Fanuc TP program (LS listing): UP022.LS

/PROG  UP022
/ATTR
OWNER		= GME;
COMMENT		= "Soldadura Est.";
PROG_SIZE	= 16158;
CREATE		= DATE 17-04-05  TIME 12:29:44;
MODIFIED	= DATE 24-03-02  TIME 05:16:32;
FILE_NAME	= UP022;
VERSION		= 0;
LINE_COUNT	= 65;
MEMORY_SIZE	= 30858;
PROTECT		= READ_WRITE;
TCD:  STACK_SIZE	= 500,
      TASK_PRIORITY	= 50,
      TIME_SLICE	= 0,
      BUSY_LAMP_OFF	= 0,
      ABORT_REQUEST	= 0,
      PAUSE_REQUEST	= 0;
DEFAULT_GROUP	= 1,1,1,1,*;
CONTROL_CODE	= 00000001 00000000;
/APPL
/MN
   1:  UFRAME_NUM=1 ;
   2:  UTOOL_NUM=2 ;
   3:  PAYLOAD[2] ;
   4:J P[1] 100% CNT0 ACC100 TB    .10sec,P-SPS    ;
      1:  TC_ONLINE (ON) ;
      2:  DO[23]=(OFF) ;
      3:  DO[16]=(ON) ;
      4:  TIMER[4]=RESET ;
      5:  TIMER[4]=START ;
      6:  CALL MAKRO050    ;
      7:  !Lib. de Herramientas ;
      8:  DO[80]=ON ;
      9:  DO[79]=ON ;
     10:  DO[78]=OFF ;
     11:  DO[77]=OFF ;
     12:  DO[76]=ON ;
     13:  DO[74]=OFF ;
     14:  !Lib. de Anticolisiones ;
     15:  DO[43]=ON ;
     16:  DO[44]=ON ;
     17:  DO[45]=ON ;
     18:  DO[46]=ON ;
     19:  DO[47]=ON ;
     20:  DO[48]=ON ;
     21:  !Apagar Pos. Base ;
     22:  DO[15]=OFF ;
     23:  !Robot en Trayectoria ;
     24:  DO[16]=ON ;
     25:  !Basculante 1 en Pos. de Reposo ;
     26:  IF (!DI[842] AND DO[12]),CALL MAKRO072 ;
     27:  WAIT (M[96])    ;
     28:  WAIT (DI[23])    ;
     29:  DO[23]=ON ;
     30:  TC_ONLINE (M[1] AND M[30] AND M[31] AND M[34] AND M[95] AND M[96]) ;
       ------ ;
   5:J P[2] 100% CNT100 ACC100 TB   0.00sec,P-SPS    ;
      1:  TC_ONLINE (M[1] AND M[30] AND M[31] AND M[34] AND M[95] AND M[96]) ;
       ------ ;
   6:J P[3] 100% CNT100 ACC100 TB   0.00sec,P-SPS    ;
      1:  TC_ONLINE (M[1] AND M[30] AND M[31] AND M[34] AND M[95] AND M[96]) ;
       ------ ;
   7:J P[4] 100% CNT100 ACC100 TB   0.00sec,P-SPS    ;
      1:  TC_ONLINE (M[1] AND M[30] AND M[31] AND M[34] AND M[95] AND M[96]) ;
       ------ ;
   8:  !5qa802035b_007_gps0005_L ;
   9:  !Punto de Sol. No. 10044 ;
  10:J P[5] 100% CNT0 ACC100 TB    .10sec,P-SPS Offset,PR[11]    ;
      1:  TC_ONLINE (ON) ;
      2:  DO[23]=(OFF) ;
      3:  WAIT (!DI[16] AND DI[23])    ;
      4:  CALL VW_USER(Basic1,EZSP,Nr1,ProgNr=99, , ,S-Punkt=10044,Fzg_Typ=7,EIN/AUS=ON) ;
      5:  GO[2]=(R[197]+10) ;
      6:  WAIT (!DI[129] OR DI[26])    ;
      7:  CALL MAKRO080    ;
      8:  WAIT (DI[23])    ;
      9:  DO[23]=(ON) ;
     10:  TC_ONLINE (M[1] AND M[30] AND M[31] AND M[34] AND M[95] AND M[96]) ;
       ------ ;
  11:J P[6] 100% CNT100 ACC100 TB   0.00sec,P-SPS    ;
      1:  TC_ONLINE (M[1] AND M[30] AND M[31] AND M[34] AND M[95] AND M[96]) ;
       ------ ;
  12:J P[7] 100% CNT100 ACC100 TB   0.00sec,P-SPS    ;
      1:  TC_ONLINE (M[1] AND M[30] AND M[31] AND M[34] AND M[95] AND M[96]) ;
       ------ ;
  13:J P[8] 100% CNT100 ACC100 TB   0.00sec,P-SPS    ;
      1:  TC_ONLINE (M[1] AND M[30] AND M[31] AND M[34] AND M[95] AND M[96]) ;
       ------ ;
  14:J P[9] 100% CNT100 ACC100 TB   0.00sec,P-SPS    ;
      1:  TC_ONLINE (M[1] AND M[30] AND M[31] AND M[34] AND M[95] AND M[96]) ;
       ------ ;
  15:  !5qa802035b_007_gps0007_L ;
  16:  !Punto de Sol. No. 10045 ;
  17:J P[10] 100% CNT0 ACC100 TB    .10sec,P-SPS Offset,PR[11]    ;
      1:  TC_ONLINE (ON) ;
      2:  DO[23]=(OFF) ;
      3:  WAIT (!DI[16] AND DI[23])    ;
      4:  CALL VW_USER(Basic1,EZSP,Nr1,ProgNr=99, , ,S-Punkt=10045,Fzg_Typ=7,EIN/AUS=ON) ;
      5:  GO[2]=(R[197]) ;
      6:  WAIT (!DI[129] OR DI[26])    ;
      7:  CALL MAKRO080    ;
      8:  WAIT (DI[23])    ;
      9:  DO[23]=(ON) ;
     10:  TC_ONLINE (M[1] AND M[30] AND M[31] AND M[34] AND M[95] AND M[96]) ;
       ------ ;
  18:J P[11] 100% CNT100 ACC100 TB   0.00sec,P-SPS    ;
      1:  TC_ONLINE (M[1] AND M[30] AND M[31] AND M[34] AND M[95] AND M[96]) ;
       ------ ;
  19:  !5qa802035b_023_xps0004_L ;
  20:  !Punto de Sol. No. 10046 ;
  21:J P[12] 100% CNT0 ACC100 TB    .10sec,P-SPS Offset,PR[11]    ;
      1:  TC_ONLINE (ON) ;
      2:  DO[23]=(OFF) ;
      3:  WAIT (!DI[16] AND DI[23])    ;
      4:  CALL VW_USER(Basic1,EZSP,Nr1,ProgNr=99, , ,S-Punkt=10046,Fzg_Typ=7,EIN/AUS=ON) ;
      5:  GO[2]=(R[197]+5) ;
      6:  WAIT (!DI[129] OR DI[26])    ;
      7:  CALL MAKRO080    ;
      8:  WAIT (DI[23])    ;
      9:  DO[23]=(ON) ;
     10:  TC_ONLINE (M[1] AND M[30] AND M[31] AND M[34] AND M[95] AND M[96]) ;
       ------ ;
  22:J P[13] 100% CNT100 ACC100 TB   0.00sec,P-SPS    ;
      1:  TC_ONLINE (M[1] AND M[30] AND M[31] AND M[34] AND M[95] AND M[96]) ;
       ------ ;
  23:J P[14] 100% CNT100 ACC100 TB   0.00sec,P-SPS    ;
      1:  TC_ONLINE (M[1] AND M[30] AND M[31] AND M[34] AND M[95] AND M[96]) ;
       ------ ;
  24:J P[15] 100% CNT100 ACC100 TB   0.00sec,P-SPS    ;
      1:  TC_ONLINE (M[1] AND M[30] AND M[31] AND M[34] AND M[95] AND M[96]) ;
       ------ ;
  25:J P[16] 100% CNT100 ACC100 TB   0.00sec,P-SPS    ;
      1:  TC_ONLINE (M[1] AND M[30] AND M[31] AND M[34] AND M[95] AND M[96]) ;
       ------ ;
  26:J P[17] 100% CNT100 ACC100 TB   0.00sec,P-SPS    ;
      1:  TC_ONLINE (M[1] AND M[30] AND M[31] AND M[34] AND M[95] AND M[96]) ;
       ------ ;
  27:J P[18] 100% CNT100 ACC100 TB   0.00sec,P-SPS    ;
      1:  TC_ONLINE (M[1] AND M[30] AND M[31] AND M[34] AND M[95] AND M[96]) ;
       ------ ;
  28:J P[19] 100% CNT100 ACC100 TB   0.00sec,P-SPS    ;
      1:  TC_ONLINE (M[1] AND M[30] AND M[31] AND M[34] AND M[95] AND M[96]) ;
       ------ ;
  29:  !5qa802035b_013_nps0004_L ;
  30:  !Punto de Sol. No. 10053 ;
  31:J P[20] 100% CNT0 ACC100 TB    .10sec,P-SPS Offset,PR[11]    ;
      1:  TC_ONLINE (ON) ;
      2:  DO[23]=(OFF) ;
      3:  WAIT (!DI[16] AND DI[23])    ;
      4:  CALL VW_USER(Basic1,EZSP,Nr1,ProgNr=99, , ,S-Punkt=10053,Fzg_Typ=7,EIN/AUS=ON) ;
      5:  GO[2]=(R[197]) ;
      6:  WAIT (!DI[129] OR DI[26])    ;
      7:  CALL MAKRO080    ;
      8:  WAIT (DI[23])    ;
      9:  DO[23]=(ON) ;
     10:  TC_ONLINE (M[1] AND M[30] AND M[31] AND M[34] AND M[95] AND M[96]) ;
       ------ ;
  32:  !5qa802035b_013_nps0003_L ;
  33:  !Punto de Sol. No. 10052 ;
  34:J P[21] 100% CNT0 ACC100 TB    .10sec,P-SPS Offset,PR[11]    ;
      1:  TC_ONLINE (ON) ;
      2:  DO[23]=(OFF) ;
      3:  WAIT (!DI[16] AND DI[23])    ;
      4:  CALL VW_USER(Basic1,EZSP,Nr1,ProgNr=99, , ,S-Punkt=10052,Fzg_Typ=7,EIN/AUS=ON) ;
      5:  GO[2]=(R[197]+10) ;
      6:  WAIT (!DI[129] OR DI[26])    ;
      7:  CALL MAKRO080    ;
      8:  WAIT (DI[23])    ;
      9:  DO[23]=(ON) ;
     10:  TC_ONLINE (M[1] AND M[30] AND M[31] AND M[34] AND M[95] AND M[96]) ;
       ------ ;
  35:J P[22] 100% CNT100 ACC100 TB   0.00sec,P-SPS    ;
      1:  TC_ONLINE (M[1] AND M[30] AND M[31] AND M[34] AND M[95] AND M[96]) ;
       ------ ;
  36:J P[23] 100% CNT100 ACC100 TB   0.00sec,P-SPS    ;
      1:  TC_ONLINE (M[1] AND M[30] AND M[31] AND M[34] AND M[95] AND M[96]) ;
       ------ ;
  37:  !5qa802035b_029_adps0008_L ;
  38:  !Punto de Sol. No. 10051 ;
  39:J P[24] 100% CNT0 ACC100 TB    .10sec,P-SPS Offset,PR[11]    ;
      1:  TC_ONLINE (ON) ;
      2:  DO[23]=(OFF) ;
      3:  WAIT (!DI[16] AND DI[23])    ;
      4:  CALL VW_USER(Basic1,EZSP,Nr1,ProgNr=99, , ,S-Punkt=10051,Fzg_Typ=7,EIN/AUS=ON) ;
      5:  GO[2]=(R[197]) ;
      6:  WAIT (!DI[129] OR DI[26])    ;
      7:  CALL MAKRO080    ;
      8:  WAIT (DI[23])    ;
      9:  DO[23]=(ON) ;
     10:  TC_ONLINE (M[1] AND M[30] AND M[31] AND M[34] AND M[95] AND M[96]) ;
       ------ ;
  40:J P[25] 100% CNT100 ACC100 TB   0.00sec,P-SPS    ;
      1:  TC_ONLINE (M[1] AND M[30] AND M[31] AND M[34] AND M[95] AND M[96]) ;
       ------ ;
  41:  !5qa802035b_029_adps0009_L ;
  42:  !Punto de Sol. No. 10050 ;
  43:J P[26] 100% CNT0 ACC100 TB    .10sec,P-SPS Offset,PR[11]    ;
      1:  TC_ONLINE (ON) ;
      2:  DO[23]=(OFF) ;
      3:  WAIT (!DI[16] AND DI[23])    ;
      4:  CALL VW_USER(Basic1,EZSP,Nr1,ProgNr=99, , ,S-Punkt=10050,Fzg_Typ=7,EIN/AUS=ON) ;
      5:  GO[2]=(R[197]) ;
      6:  WAIT (!DI[129] OR DI[26])    ;
      7:  CALL MAKRO080    ;
      8:  WAIT (DI[23])    ;
      9:  DO[23]=(ON) ;
     10:  TC_ONLINE (M[1] AND M[30] AND M[31] AND M[34] AND M[95] AND M[96]) ;
       ------ ;
  44:  !5qa802035b_029_adps0005_L ;
  45:  !Punto de Sol. No. 10049 ;
  46:J P[27] 100% CNT0 ACC100 TB    .10sec,P-SPS Offset,PR[11]    ;
      1:  TC_ONLINE (ON) ;
      2:  DO[23]=(OFF) ;
      3:  WAIT (!DI[16] AND DI[23])    ;
      4:  CALL VW_USER(Basic1,EZSP,Nr1,ProgNr=99, , ,S-Punkt=10049,Fzg_Typ=7,EIN/AUS=ON) ;
      5:  GO[2]=(R[197]) ;
      6:  WAIT (!DI[129] OR DI[26])    ;
      7:  CALL MAKRO080    ;
      8:  WAIT (DI[23])    ;
      9:  DO[23]=(ON) ;
     10:  TC_ONLINE (M[1] AND M[30] AND M[31] AND M[34] AND M[95] AND M[96]) ;
       ------ ;
  47:J P[28] 100% CNT100 ACC100 TB   0.00sec,P-SPS    ;
      1:  TC_ONLINE (M[1] AND M[30] AND M[31] AND M[34] AND M[95] AND M[96]) ;
       ------ ;
  48:  !5qa802035b_013_nps0002_L ;
  49:  !Punto de Sol. No. 10048 ;
  50:J P[29] 100% CNT0 ACC100 TB    .10sec,P-SPS Offset,PR[11]    ;
      1:  TC_ONLINE (ON) ;
      2:  DO[23]=(OFF) ;
      3:  WAIT (!DI[16] AND DI[23])    ;
      4:  CALL VW_USER(Basic1,EZSP,Nr1,ProgNr=99, , ,S-Punkt=10048,Fzg_Typ=7,EIN/AUS=ON) ;
      5:  GO[2]=(R[197]) ;
      6:  WAIT (!DI[129] OR DI[26])    ;
      7:  CALL MAKRO080    ;
      8:  WAIT (DI[23])    ;
      9:  DO[23]=(ON) ;
     10:  TC_ONLINE (M[1] AND M[30] AND M[31] AND M[34] AND M[95] AND M[96]) ;
       ------ ;
  51:  !5qa802035b_013_nps0001_L ;
  52:  !Punto de Sol. No. 10047 ;
  53:J P[30] 100% CNT0 ACC100 TB    .10sec,P-SPS Offset,PR[11]    ;
      1:  TC_ONLINE (ON) ;
      2:  DO[23]=(OFF) ;
      3:  WAIT (!DI[16] AND DI[23])    ;
      4:  CALL VW_USER(Basic1,EZSP,Nr1,ProgNr=99, , ,S-Punkt=10047,Fzg_Typ=7,EIN/AUS=ON) ;
      5:  GO[2]=(R[197]) ;
      6:  WAIT (!DI[129] OR DI[26])    ;
      7:  CALL MAKRO080    ;
      8:  WAIT (DI[23])    ;
      9:  DO[23]=(ON) ;
     10:  TC_ONLINE (M[1] AND M[30] AND M[31] AND M[34] AND M[95] AND M[96]) ;
       ------ ;
  54:J P[31] 100% CNT100 ACC100 TB   0.00sec,P-SPS    ;
      1:  TC_ONLINE (M[1] AND M[30] AND M[31] AND M[34] AND M[95] AND M[96]) ;
       ------ ;
  55:J P[32] 100% CNT100 ACC100 TB   0.00sec,P-SPS    ;
      1:  TC_ONLINE (M[1] AND M[30] AND M[31] AND M[34] AND M[95] AND M[96]) ;
       ------ ;
  56:J P[33] 100% CNT100 ACC100 TB   0.00sec,P-SPS    ;
      1:  TC_ONLINE (M[1] AND M[30] AND M[31] AND M[34] AND M[95] AND M[96]) ;
       ------ ;
  57:J P[34] 100% CNT100 ACC100 TB   0.00sec,P-SPS    ;
      1:  TC_ONLINE (M[1] AND M[30] AND M[31] AND M[34] AND M[95] AND M[96]) ;
       ------ ;
  58:J P[35] 100% CNT100 ACC100 TB   0.00sec,P-SPS    ;
      1:  TC_ONLINE (M[1] AND M[30] AND M[31] AND M[34] AND M[95] AND M[96]) ;
       ------ ;
  59:  !5qa802035b_007_gps0003_L ;
  60:  !Punto de Sol. No. 10054 ;
  61:  !Fin de Trabajo 2 ;
  62:J P[36] 100% CNT0 ACC100 TB    .10sec,P-SPS Offset,PR[11]    ;
      1:  TC_ONLINE (ON) ;
      2:  DO[23]=(OFF) ;
      3:  WAIT (!DI[16] AND DI[23])    ;
      4:  CALL VW_USER(Basic1,EZSP,Nr1,ProgNr=99, , ,S-Punkt=10054,Fzg_Typ=7,EIN/AUS=ON) ;
      5:  GO[2]=(R[197]) ;
      6:  WAIT (!DI[129] OR DI[26])    ;
      7:  CALL MAKRO080    ;
      8:  IF (!DI[145] AND !DI[129]),CALL MAKRO002 ;
      9:  WAIT (DI[23])    ;
     10:  DO[23]=(ON) ;
     11:  TC_ONLINE (M[1] AND M[30] AND M[31] AND M[34] AND M[95] AND M[96]) ;
       ------ ;
  63:J P[37] 100% CNT100 ACC100 TB   0.00sec,P-SPS    ;
      1:  TC_ONLINE (M[1] AND M[30] AND M[31] AND M[34] AND M[95] AND M[96]) ;
       ------ ;
  64:J P[38] 100% CNT100 ACC100 TB   0.00sec,P-SPS    ;
      1:  TC_ONLINE (M[1] AND M[30] AND M[31] AND M[34] AND M[95] AND M[96]) ;
       ------ ;
  65:J P[39] 100% CNT0 ACC100 TB    .10sec,P-SPS    ;
      1:  TC_ONLINE (ON) ;
      2:  DO[23]=(OFF) ;
      3:  TIMER[4]=STOP ;
      4:  WAIT (DI[23])    ;
      5:  CALL VW_USER(Basic1,EZSP,Nr1 Service,ProgNr=31, , ,S-Punkt=31, ,EIN/AUS=1) ;
      6:  DO[23]=(ON) ;
      7:  TC_ONLINE (M[1] AND M[30] AND M[31] AND M[34] AND M[95] AND M[96]) ;
       ------ ;
/POS
P[1]{
   GP1:
	UF : 1, UT : 2,		CONFIG : 'N U T, 0, 0, 0',
	RX =  1133.105  mm,	RY =   304.802  mm,	RZ =  -956.232  mm,
	RW =    13.347 deg,	RP =    14.205 deg,	RR =   -95.327 deg
   GP2:
	UF : 1, UT : 2,
	J1=   100.000  mm
   GP3:
	UF : 1, UT : 2,
	J1=     0.000  mm
   GP4:
	UF : 1, UT : 2,
	J1=     0.000  mm
};
P[2]{
   GP1:
	UF : 1, UT : 2,		CONFIG : 'N U T, 0, 0, 0',
	RX =    66.244  mm,	RY = -1097.752  mm,	RZ =  -631.601  mm,
	RW =     4.264 deg,	RP =    -9.468 deg,	RR =  -138.417 deg
   GP2:
	UF : 1, UT : 2,
	J1=   120.000  mm
   GP3:
	UF : 1, UT : 2,
	J1=     0.000  mm
   GP4:
	UF : 1, UT : 2,
	J1=     0.000  mm
};
P[3]{
   GP1:
	UF : 1, UT : 2,		CONFIG : 'F U T, 0, 0, 0',
	RX =  -363.159  mm,	RY =  -637.383  mm,	RZ =   295.420  mm,
	RW =   171.646 deg,	RP =   -81.600 deg,	RR =    73.386 deg
   GP2:
	UF : 1, UT : 2,
	J1=   100.000  mm
   GP3:
	UF : 1, UT : 2,
	J1=     0.000  mm
   GP4:
	UF : 1, UT : 2,
	J1=     0.000  mm
};
P[4]{
   GP1:
	UF : 1, UT : 2,		CONFIG : 'F U T, 0, 0, 0',
	RX =  -355.700  mm,	RY =  -477.893  mm,	RZ =   268.172  mm,
	RW =   171.646 deg,	RP =   -81.600 deg,	RR =    73.385 deg
   GP2:
	UF : 1, UT : 2,
	J1=   100.000  mm
   GP3:
	UF : 1, UT : 2,
	J1=     0.000  mm
   GP4:
	UF : 1, UT : 2,
	J1=     0.000  mm
};
P[5]{
   GP1:
	UF : 1, UT : 2,		CONFIG : 'F U T, 0, 0, 0',
	RX =  -357.224  mm,	RY =  -466.560  mm,	RZ =   272.864  mm,
	RW =   169.052 deg,	RP =   -83.613 deg,	RR =    76.002 deg
   GP2:
	UF : 1, UT : 2,
	J1=    30.200  mm
   GP3:
	UF : 1, UT : 2,
	J1=     0.000  mm
   GP4:
	UF : 1, UT : 2,
	J1=     0.000  mm
};
P[6]{
   GP1:
	UF : 1, UT : 2,		CONFIG : 'F U T, 0, 0, 0',
	RX =  -359.183  mm,	RY =  -476.278  mm,	RZ =   268.090  mm,
	RW =   171.646 deg,	RP =   -81.600 deg,	RR =    73.386 deg
   GP2:
	UF : 1, UT : 2,
	J1=   100.000  mm
   GP3:
	UF : 1, UT : 2,
	J1=     0.000  mm
   GP4:
	UF : 1, UT : 2,
	J1=     0.000  mm
};
P[7]{
   GP1:
	UF : 1, UT : 2,		CONFIG : 'F U T, 0, 0, 0',
	RX =  -362.737  mm,	RY =  -548.013  mm,	RZ =   274.263  mm,
	RW =   171.645 deg,	RP =   -81.600 deg,	RR =    73.386 deg
   GP2:
	UF : 1, UT : 2,
	J1=   100.000  mm
   GP3:
	UF : 1, UT : 2,
	J1=     0.000  mm
   GP4:
	UF : 1, UT : 2,
	J1=     0.000  mm
};
P[8]{
   GP1:
	UF : 1, UT : 2,		CONFIG : 'F U T, 0, 0, 0',
	RX =  -129.372  mm,	RY =  -655.590  mm,	RZ =   283.757  mm,
	RW =   171.646 deg,	RP =   -81.600 deg,	RR =    73.386 deg
   GP2:
	UF : 1, UT : 2,
	J1=   100.000  mm
   GP3:
	UF : 1, UT : 2,
	J1=     0.000  mm
   GP4:
	UF : 1, UT : 2,
	J1=     0.000  mm
};
P[9]{
   GP1:
	UF : 1, UT : 2,		CONFIG : 'F U T, 0, 0, 0',
	RX =  -130.559  mm,	RY =  -455.743  mm,	RZ =   264.260  mm,
	RW =   177.915 deg,	RP =   -81.600 deg,	RR =    73.387 deg
   GP2:
	UF : 1, UT : 2,
	J1=   100.000  mm
   GP3:
	UF : 1, UT : 2,
	J1=     0.000  mm
   GP4:
	UF : 1, UT : 2,
	J1=     0.000  mm
};
P[10]{
   GP1:
	UF : 1, UT : 2,		CONFIG : 'F U T, 0, 0, 0',
	RX =  -129.044  mm,	RY =  -454.645  mm,	RZ =   269.211  mm,
	RW =   177.993 deg,	RP =   -81.609 deg,	RR =    73.315 deg
   GP2:
	UF : 1, UT : 2,
	J1=    27.704  mm
   GP3:
	UF : 1, UT : 2,
	J1=     0.000  mm
   GP4:
	UF : 1, UT : 2,
	J1=     0.000  mm
};
P[11]{
   GP1:
	UF : 1, UT : 2,		CONFIG : 'F U T, 0, 0, 0',
	RX =   -90.615  mm,	RY =  -443.457  mm,	RZ =   251.615  mm,
	RW =  -142.266 deg,	RP =   -79.369 deg,	RR =    33.067 deg
   GP2:
	UF : 1, UT : 2,
	J1=    40.000  mm
   GP3:
	UF : 1, UT : 2,
	J1=     0.000  mm
   GP4:
	UF : 1, UT : 2,
	J1=     0.000  mm
};
P[12]{
   GP1:
	UF : 1, UT : 2,		CONFIG : 'F U T, 0, 0, 0',
	RX =   -68.121  mm,	RY =  -445.925  mm,	RZ =   268.522  mm,
	RW =  -161.036 deg,	RP =   -72.891 deg,	RR =    52.407 deg
   GP2:
	UF : 1, UT : 2,
	J1=    22.000  mm
   GP3:
	UF : 1, UT : 2,
	J1=     0.000  mm
   GP4:
	UF : 1, UT : 2,
	J1=     0.000  mm
};
P[13]{
   GP1:
	UF : 1, UT : 2,		CONFIG : 'F U T, 0, 0, 0',
	RX =   -75.083  mm,	RY =  -452.168  mm,	RZ =   267.964  mm,
	RW =  -166.090 deg,	RP =   -74.801 deg,	RR =    57.641 deg
   GP2:
	UF : 1, UT : 2,
	J1=   100.000  mm
   GP3:
	UF : 1, UT : 2,
	J1=     0.000  mm
   GP4:
	UF : 1, UT : 2,
	J1=     0.000  mm
};
P[14]{
   GP1:
	UF : 1, UT : 2,		CONFIG : 'F U T, 0, 0, 0',
	RX =  -106.428  mm,	RY =  -546.571  mm,	RZ =   283.041  mm,
	RW =  -166.090 deg,	RP =   -74.801 deg,	RR =    57.641 deg
   GP2:
	UF : 1, UT : 2,
	J1=   100.000  mm
   GP3:
	UF : 1, UT : 2,
	J1=     0.000  mm
   GP4:
	UF : 1, UT : 2,
	J1=     0.000  mm
};
P[15]{
   GP1:
	UF : 1, UT : 2,		CONFIG : 'F U T, 0, 0, 0',
	RX =   -58.763  mm,	RY =  -675.997  mm,	RZ =   305.810  mm,
	RW =  -154.703 deg,	RP =   -81.518 deg,	RR =    46.029 deg
   GP2:
	UF : 1, UT : 2,
	J1=   100.000  mm
   GP3:
	UF : 1, UT : 2,
	J1=     0.000  mm
   GP4:
	UF : 1, UT : 2,
	J1=     0.000  mm
};
P[16]{
   GP1:
	UF : 1, UT : 2,		CONFIG : 'F U T, 0, 0, 0',
	RX =   167.422  mm,	RY =  -755.632  mm,	RZ =   268.835  mm,
	RW =  -117.579 deg,	RP =   -78.602 deg,	RR =     8.529 deg
   GP2:
	UF : 1, UT : 2,
	J1=   100.000  mm
   GP3:
	UF : 1, UT : 2,
	J1=     0.000  mm
   GP4:
	UF : 1, UT : 2,
	J1=     0.000  mm
};
P[17]{
   GP1:
	UF : 1, UT : 2,		CONFIG : 'F U T, 0, 0, 0',
	RX =   224.739  mm,	RY =  -491.620  mm,	RZ =   -22.031  mm,
	RW =  -102.440 deg,	RP =   -64.865 deg,	RR =    -7.291 deg
   GP2:
	UF : 1, UT : 2,
	J1=   100.000  mm
   GP3:
	UF : 1, UT : 2,
	J1=     0.000  mm
   GP4:
	UF : 1, UT : 2,
	J1=     0.000  mm
};
P[18]{
   GP1:
	UF : 1, UT : 2,		CONFIG : 'F U T, 0, 0, 0',
	RX =   186.154  mm,	RY =  -445.858  mm,	RZ =     4.056  mm,
	RW =  -100.027 deg,	RP =   -58.299 deg,	RR =   -10.029 deg
   GP2:
	UF : 1, UT : 2,
	J1=   100.000  mm
   GP3:
	UF : 1, UT : 2,
	J1=     0.000  mm
   GP4:
	UF : 1, UT : 2,
	J1=     0.000  mm
};
P[19]{
   GP1:
	UF : 1, UT : 2,		CONFIG : 'F U T, 0, 0, 0',
	RX =   173.095  mm,	RY =  -434.006  mm,	RZ =    19.013  mm,
	RW =  -106.388 deg,	RP =   -56.239 deg,	RR =    -2.521 deg
   GP2:
	UF : 1, UT : 2,
	J1=   100.000  mm
   GP3:
	UF : 1, UT : 2,
	J1=     0.000  mm
   GP4:
	UF : 1, UT : 2,
	J1=     0.000  mm
};
P[20]{
   GP1:
	UF : 1, UT : 2,		CONFIG : 'F U T, 0, 0, 0',
	RX =   175.846  mm,	RY =  -432.191  mm,	RZ =    12.536  mm,
	RW =  -108.251 deg,	RP =   -55.844 deg,	RR =     -.274 deg
   GP2:
	UF : 1, UT : 2,
	J1=    22.000  mm
   GP3:
	UF : 1, UT : 2,
	J1=     0.000  mm
   GP4:
	UF : 1, UT : 2,
	J1=     0.000  mm
};
P[21]{
   GP1:
	UF : 1, UT : 2,		CONFIG : 'F U T, 0, 0, 0',
	RX =   165.490  mm,	RY =  -431.087  mm,	RZ =    21.456  mm,
	RW =  -105.966 deg,	RP =   -56.296 deg,	RR =    -2.622 deg
   GP2:
	UF : 1, UT : 2,
	J1=    20.700  mm
   GP3:
	UF : 1, UT : 2,
	J1=     0.000  mm
   GP4:
	UF : 1, UT : 2,
	J1=     0.000  mm
};
P[22]{
   GP1:
	UF : 1, UT : 2,		CONFIG : 'F U T, 0, 0, 0',
	RX =   154.830  mm,	RY =  -426.794  mm,	RZ =    23.878  mm,
	RW =  -103.158 deg,	RP =   -56.239 deg,	RR =    -2.521 deg
   GP2:
	UF : 1, UT : 2,
	J1=    30.000  mm
   GP3:
	UF : 1, UT : 2,
	J1=     0.000  mm
   GP4:
	UF : 1, UT : 2,
	J1=     0.000  mm
};
P[23]{
   GP1:
	UF : 1, UT : 2,		CONFIG : 'F U T, 0, 0, 0',
	RX =   126.370  mm,	RY =  -417.423  mm,	RZ =    43.158  mm,
	RW =   -98.232 deg,	RP =   -56.239 deg,	RR =    -2.521 deg
   GP2:
	UF : 1, UT : 2,
	J1=    19.500  mm
   GP3:
	UF : 1, UT : 2,
	J1=     0.000  mm
   GP4:
	UF : 1, UT : 2,
	J1=     0.000  mm
};
P[24]{
   GP1:
	UF : 1, UT : 2,		CONFIG : 'F U T, 0, 0, 0',
	RX =   124.011  mm,	RY =  -422.950  mm,	RZ =    44.190  mm,
	RW =  -102.498 deg,	RP =   -54.643 deg,	RR =     2.578 deg
   GP2:
	UF : 1, UT : 2,
	J1=    22.000  mm
   GP3:
	UF : 1, UT : 2,
	J1=     0.000  mm
   GP4:
	UF : 1, UT : 2,
	J1=     0.000  mm
};
P[25]{
   GP1:
	UF : 1, UT : 2,		CONFIG : 'F U T, 0, 0, 0',
	RX =   107.911  mm,	RY =  -418.925  mm,	RZ =    49.571  mm,
	RW =   -97.335 deg,	RP =   -56.035 deg,	RR =     -.254 deg
   GP2:
	UF : 1, UT : 2,
	J1=    21.400  mm
   GP3:
	UF : 1, UT : 2,
	J1=     0.000  mm
   GP4:
	UF : 1, UT : 2,
	J1=     0.000  mm
};
P[26]{
   GP1:
	UF : 1, UT : 2,		CONFIG : 'F U T, 0, 0, 0',
	RX =   105.438  mm,	RY =  -411.916  mm,	RZ =    56.428  mm,
	RW =   -99.772 deg,	RP =   -55.781 deg,	RR =     2.693 deg
   GP2:
	UF : 1, UT : 2,
	J1=    22.000  mm
   GP3:
	UF : 1, UT : 2,
	J1=     0.000  mm
   GP4:
	UF : 1, UT : 2,
	J1=     0.000  mm
};
P[27]{
   GP1:
	UF : 1, UT : 2,		CONFIG : 'F U T, 0, 0, 0',
	RX =   124.880  mm,	RY =  -410.640  mm,	RZ =    42.285  mm,
	RW =   -98.955 deg,	RP =   -55.878 deg,	RR =     1.712 deg
   GP2:
	UF : 1, UT : 2,
	J1=    28.308  mm
   GP3:
	UF : 1, UT : 2,
	J1=     0.000  mm
   GP4:
	UF : 1, UT : 2,
	J1=     0.000  mm
};
P[28]{
   GP1:
	UF : 1, UT : 2,		CONFIG : 'F U T, 0, 0, 0',
	RX =   140.148  mm,	RY =  -413.533  mm,	RZ =    31.554  mm,
	RW =   -97.340 deg,	RP =   -56.041 deg,	RR =     -.240 deg
   GP2:
	UF : 1, UT : 2,
	J1=    35.000  mm
   GP3:
	UF : 1, UT : 2,
	J1=     0.000  mm
   GP4:
	UF : 1, UT : 2,
	J1=     0.000  mm
};
P[29]{
   GP1:
	UF : 1, UT : 2,		CONFIG : 'F U T, 0, 0, 0',
	RX =   164.645  mm,	RY =  -412.190  mm,	RZ =    20.689  mm,
	RW =   -98.769 deg,	RP =   -56.782 deg,	RR =     1.502 deg
   GP2:
	UF : 1, UT : 2,
	J1=    22.000  mm
   GP3:
	UF : 1, UT : 2,
	J1=     0.000  mm
   GP4:
	UF : 1, UT : 2,
	J1=     0.000  mm
};
P[30]{
   GP1:
	UF : 1, UT : 2,		CONFIG : 'F U T, 0, 0, 0',
	RX =   176.762  mm,	RY =  -412.389  mm,	RZ =    12.744  mm,
	RW =   -97.537 deg,	RP =   -56.501 deg,	RR =     -.001 deg
   GP2:
	UF : 1, UT : 2,
	J1=    22.000  mm
   GP3:
	UF : 1, UT : 2,
	J1=     0.000  mm
   GP4:
	UF : 1, UT : 2,
	J1=     0.000  mm
};
P[31]{
   GP1:
	UF : 1, UT : 2,		CONFIG : 'F U T, 0, 0, 0',
	RX =   192.191  mm,	RY =  -416.396  mm,	RZ =    -5.756  mm,
	RW =   -99.853 deg,	RP =   -55.784 deg,	RR =     2.794 deg
   GP2:
	UF : 1, UT : 2,
	J1=   100.000  mm
   GP3:
	UF : 1, UT : 2,
	J1=     0.000  mm
   GP4:
	UF : 1, UT : 2,
	J1=     0.000  mm
};
P[32]{
   GP1:
	UF : 1, UT : 2,		CONFIG : 'F U T, 0, 0, 0',
	RX =   204.150  mm,	RY =  -512.716  mm,	RZ =   -10.685  mm,
	RW =   -99.853 deg,	RP =   -55.784 deg,	RR =     2.794 deg
   GP2:
	UF : 1, UT : 2,
	J1=   100.000  mm
   GP3:
	UF : 1, UT : 2,
	J1=     0.000  mm
   GP4:
	UF : 1, UT : 2,
	J1=     0.000  mm
};
P[33]{
   GP1:
	UF : 1, UT : 2,		CONFIG : 'F U T, 0, 0, 0',
	RX =   164.427  mm,	RY =  -753.815  mm,	RZ =    24.289  mm,
	RW =   -99.853 deg,	RP =   -55.784 deg,	RR =     2.794 deg
   GP2:
	UF : 1, UT : 2,
	J1=   100.000  mm
   GP3:
	UF : 1, UT : 2,
	J1=     0.000  mm
   GP4:
	UF : 1, UT : 2,
	J1=     0.000  mm
};
P[34]{
   GP1:
	UF : 1, UT : 2,		CONFIG : 'F U T, 0, 0, 0',
	RX =  -146.070  mm,	RY =  -437.528  mm,	RZ =    25.810  mm,
	RW =   -33.716 deg,	RP =     3.529 deg,	RR =  -101.420 deg
   GP2:
	UF : 1, UT : 2,
	J1=   100.000  mm
   GP3:
	UF : 1, UT : 2,
	J1=     0.000  mm
   GP4:
	UF : 1, UT : 2,
	J1=     0.000  mm
};
P[35]{
   GP1:
	UF : 1, UT : 2,		CONFIG : 'F U T, 0, 0, 0',
	RX =  -289.900  mm,	RY =  -442.594  mm,	RZ =   201.485  mm,
	RW =   -41.785 deg,	RP =     -.956 deg,	RR =   -84.186 deg
   GP2:
	UF : 1, UT : 2,
	J1=   110.000  mm
   GP3:
	UF : 1, UT : 2,
	J1=     0.000  mm
   GP4:
	UF : 1, UT : 2,
	J1=     0.000  mm
};
P[36]{
   GP1:
	UF : 1, UT : 2,		CONFIG : 'F U T, 0, 0, 0',
	RX =  -280.502  mm,	RY =  -447.089  mm,	RZ =   209.827  mm,
	RW =   -41.733 deg,	RP =     -.533 deg,	RR =   -86.310 deg
   GP2:
	UF : 1, UT : 2,
	J1=    29.717  mm
   GP3:
	UF : 1, UT : 2,
	J1=     0.000  mm
   GP4:
	UF : 1, UT : 2,
	J1=     0.000  mm
};
P[37]{
   GP1:
	UF : 1, UT : 2,		CONFIG : 'F U T, 0, 0, 0',
	RX =  -300.950  mm,	RY =  -444.366  mm,	RZ =   171.442  mm,
	RW =   -41.784 deg,	RP =     -.954 deg,	RR =   -84.186 deg
   GP2:
	UF : 1, UT : 2,
	J1=    90.559  mm
   GP3:
	UF : 1, UT : 2,
	J1=     0.000  mm
   GP4:
	UF : 1, UT : 2,
	J1=     0.000  mm
};
P[38]{
   GP1:
	UF : 1, UT : 2,		CONFIG : 'F U T, 0, 0, 0',
	RX =  -270.307  mm,	RY =  -451.727  mm,	RZ =  -454.454  mm,
	RW =   -41.784 deg,	RP =     -.954 deg,	RR =   -84.186 deg
   GP2:
	UF : 1, UT : 2,
	J1=    90.559  mm
   GP3:
	UF : 1, UT : 2,
	J1=     0.000  mm
   GP4:
	UF : 1, UT : 2,
	J1=     0.000  mm
};
P[39]{
   GP1:
	UF : 1, UT : 2,		CONFIG : 'N U T, 0, 0, 0',
	RX =  1133.105  mm,	RY =   304.802  mm,	RZ =  -956.232  mm,
	RW =    13.347 deg,	RP =    14.205 deg,	RR =   -95.327 deg
   GP2:
	UF : 1, UT : 2,
	J1=   100.000  mm
   GP3:
	UF : 1, UT : 2,
	J1=     0.000  mm
   GP4:
	UF : 1, UT : 2,
	J1=     0.000  mm
};
/END
